FUNCTION_BLOCK changeEventProcess2 (* Basic Function Block Type *)
  (* Standard: 61499-2 *)
  (* Version 0.0, 5/23/2025, azam_w, Schneider Electric, Template *)
  PACKAGE Main;
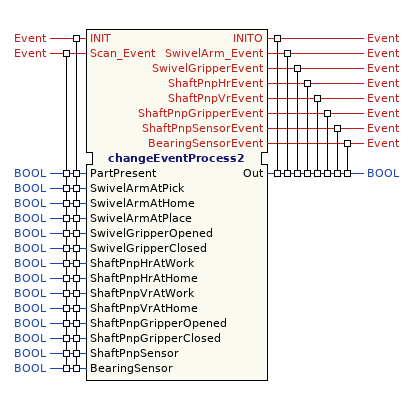
  EVENT_INPUT
    INIT WITH PartPresent, SwivelArmAtPick, SwivelArmAtHome, SwivelArmAtPlace, SwivelGripperOpened, SwivelGripperClosed, ShaftPnpHrAtWork, ShaftPnpHrAtHome, ShaftPnpVrAtWork, ShaftPnpVrAtHome, ShaftPnpGripperOpened, ShaftPnpGripperClosed, ShaftPnpSensor, BearingSensor;
    Scan_Event WITH PartPresent, SwivelArmAtPick, SwivelArmAtHome, SwivelArmAtPlace, SwivelGripperOpened, SwivelGripperClosed, ShaftPnpHrAtWork, ShaftPnpHrAtHome, ShaftPnpVrAtWork, ShaftPnpVrAtHome, ShaftPnpGripperOpened, ShaftPnpGripperClosed, ShaftPnpSensor, BearingSensor;
  END_EVENT
  EVENT_OUTPUT
    INITO WITH Out; (* Initialization Confirm *)
    SwivelArm_Event WITH Out; (* Execution Confirmation *)
    SwivelGripperEvent WITH Out;
    ShaftPnpHrEvent WITH Out;
    ShaftPnpVrEvent WITH Out;
    ShaftPnpGripperEvent WITH Out;
    ShaftPnpSensorEvent WITH Out;
    BearingSensorEvent WITH Out;
  END_EVENT
  VAR_INPUT
    PartPresent : BOOL; (* Output event qualifier *)
    SwivelArmAtPick : BOOL;
    SwivelArmAtHome : BOOL;
    SwivelArmAtPlace : BOOL;
    SwivelGripperOpened : BOOL;
    SwivelGripperClosed : BOOL;
    ShaftPnpHrAtWork : BOOL;
    ShaftPnpHrAtHome : BOOL;
    ShaftPnpVrAtWork : BOOL;
    ShaftPnpVrAtHome : BOOL;
    ShaftPnpGripperOpened : BOOL;
    ShaftPnpGripperClosed : BOOL;
    ShaftPnpSensor : BOOL;
    BearingSensor : BOOL;
  END_VAR
  VAR_OUTPUT
    Out : BOOL;
  END_VAR
  VAR
    PartPresent_PrevVAl : BOOL := FALSE;
    SwivelArmAtPick_PrevVal : BOOL := FALSE;
    SwivelArmAtHome_PrevVal : BOOL := FALSE;
    SwivelArmAtPlace_PrevVal : BOOL := FALSE;
    SwivelGripperClosed_PrevVal : BOOL;
    SwivelGripperOpened_PrevVal : BOOL;
    ShaftPnpHrAtWork_PrevVal : BOOL;
    ShaftPnpHrAtHome_PrevVal : BOOL;
    ShaftPnpVrAtWork_PrevVal : BOOL;
    ShaftPnpVrAtHome_PrevVal : BOOL;
    ShaftPnpGripperClosed_PrevVal : BOOL;
    ShaftPnpGripperOpened_PrevVal : BOOL;
    ShaftPnpSensor_PreVal : BOOL;
    BearingSensor_PreVal : BOOL;
  END_VAR
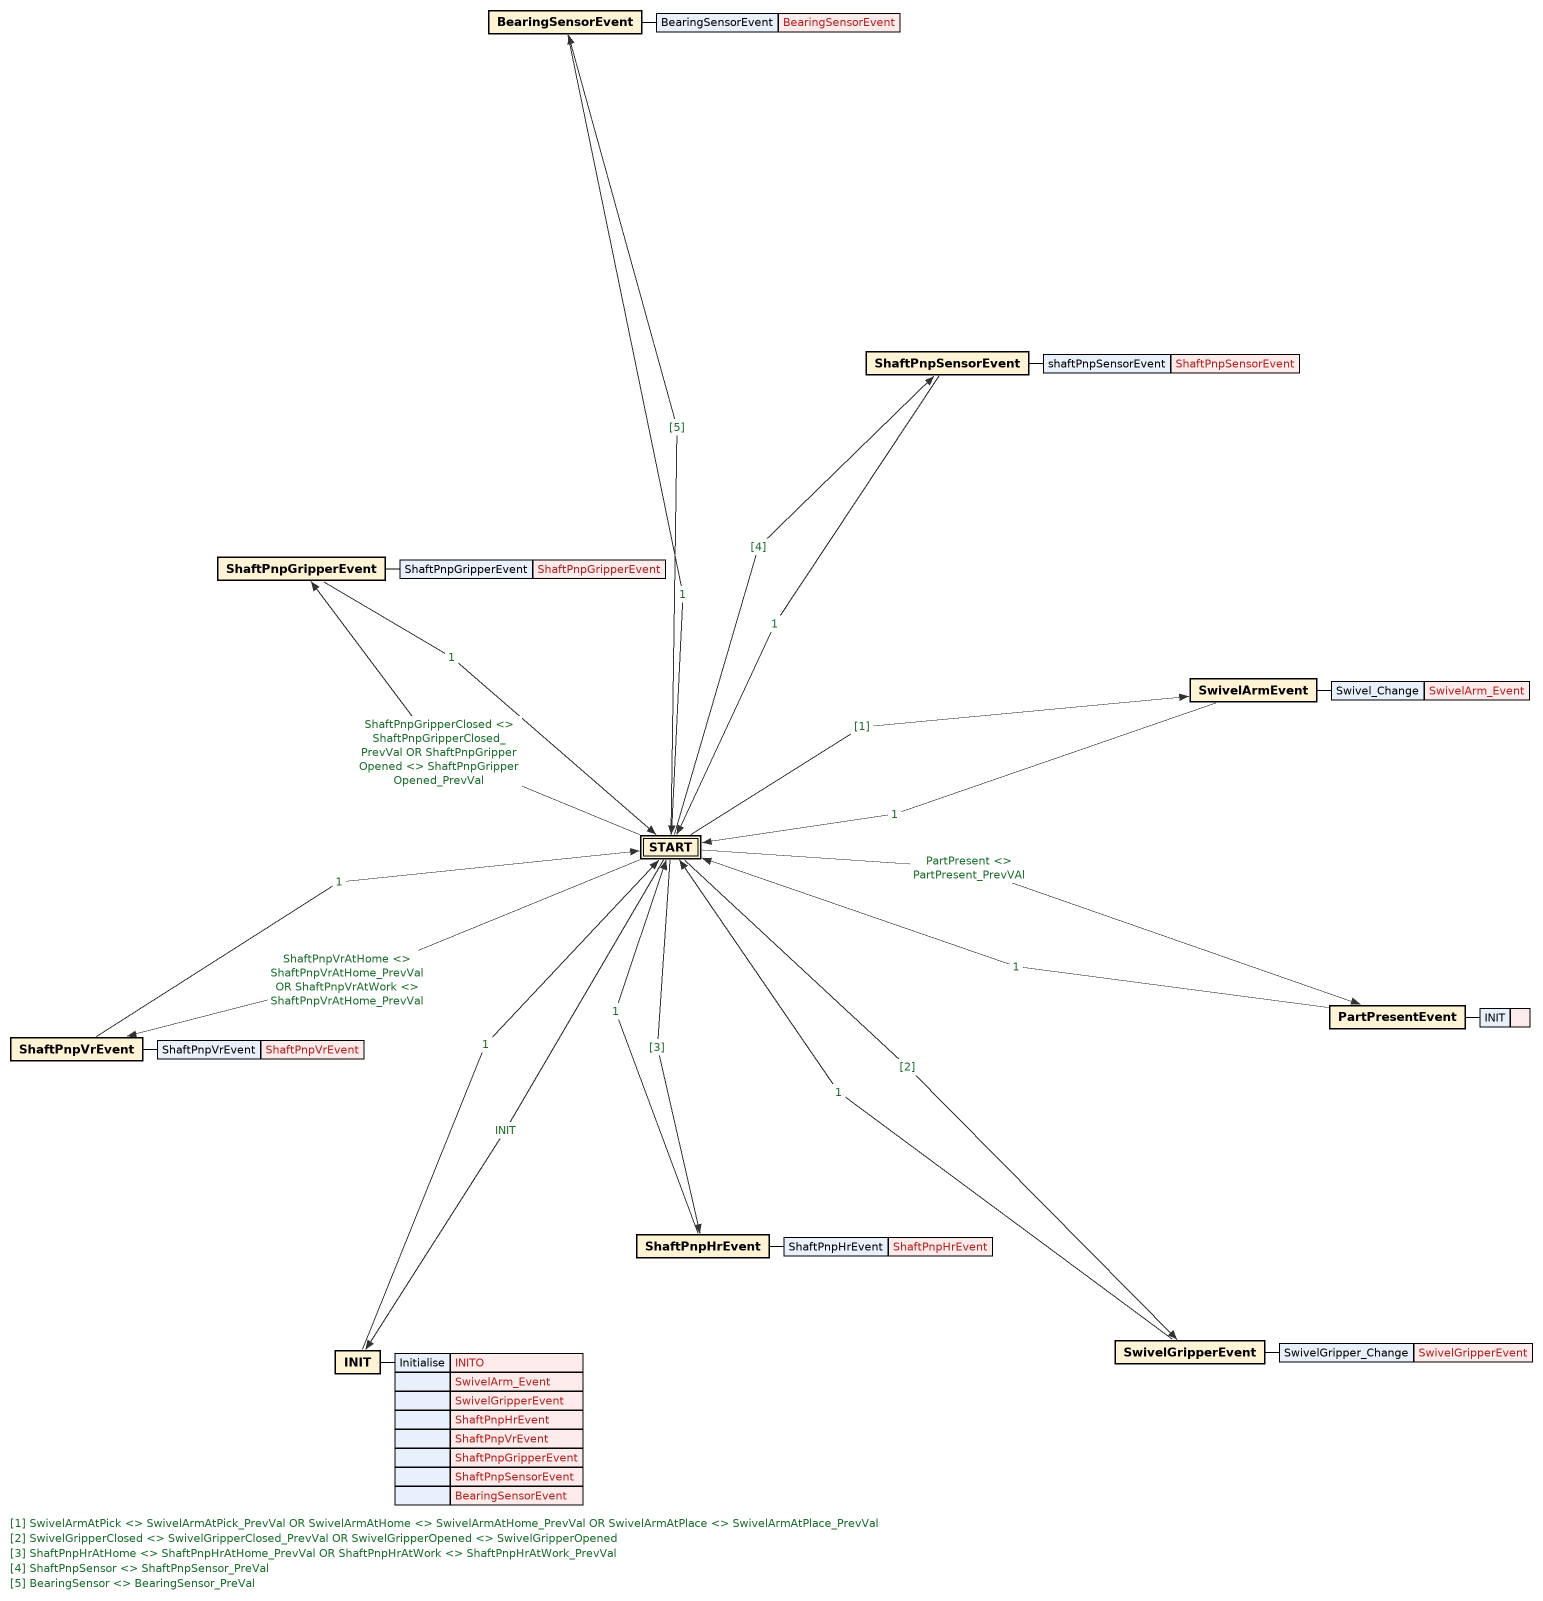
  EC_STATES
    START; (* Initial State *)
    PartPresentEvent : INIT; (* Normal execution *)
    SwivelArmEvent : Swivel_Change -> SwivelArm_Event;
    SwivelGripperEvent : SwivelGripper_Change -> SwivelGripperEvent;
    ShaftPnpHrEvent : ShaftPnpHrEvent -> ShaftPnpHrEvent;
    ShaftPnpVrEvent : ShaftPnpVrEvent -> ShaftPnpVrEvent;
    ShaftPnpGripperEvent : ShaftPnpGripperEvent -> ShaftPnpGripperEvent;
    ShaftPnpSensorEvent : shaftPnpSensorEvent -> ShaftPnpSensorEvent;
    BearingSensorEvent : BearingSensorEvent -> BearingSensorEvent;
    INIT : Initialise -> INITO, -> SwivelArm_Event, -> SwivelGripperEvent, -> ShaftPnpHrEvent, -> ShaftPnpVrEvent, -> ShaftPnpGripperEvent, -> ShaftPnpSensorEvent, -> BearingSensorEvent;
  END_STATES
  EC_TRANSITIONS
    START TO PartPresentEvent := PartPresent <> PartPresent_PrevVAl;
    PartPresentEvent TO START := 1;
    START TO SwivelArmEvent := SwivelArmAtPick <> SwivelArmAtPick_PrevVal OR SwivelArmAtHome <> SwivelArmAtHome_PrevVal OR SwivelArmAtPlace <> SwivelArmAtPlace_PrevVal;
    START TO SwivelGripperEvent := SwivelGripperClosed <> SwivelGripperClosed_PrevVal OR SwivelGripperOpened <> SwivelGripperOpened;
    SwivelGripperEvent TO START := 1;
    START TO ShaftPnpHrEvent := ShaftPnpHrAtHome <> ShaftPnpHrAtHome_PrevVal OR ShaftPnpHrAtWork <> ShaftPnpHrAtWork_PrevVal;
    ShaftPnpHrEvent TO START := 1;
    START TO ShaftPnpVrEvent := ShaftPnpVrAtHome <> ShaftPnpVrAtHome_PrevVal OR ShaftPnpVrAtWork <> ShaftPnpVrAtHome_PrevVal;
    ShaftPnpVrEvent TO START := 1;
    START TO ShaftPnpGripperEvent := ShaftPnpGripperClosed <> ShaftPnpGripperClosed_PrevVal OR ShaftPnpGripperOpened <> ShaftPnpGripperOpened_PrevVal;
    ShaftPnpGripperEvent TO START := 1;
    SwivelArmEvent TO START := 1;
    ShaftPnpSensorEvent TO START := 1;
    START TO ShaftPnpSensorEvent := ShaftPnpSensor <> ShaftPnpSensor_PreVal;
    START TO BearingSensorEvent := BearingSensor <> BearingSensor_PreVal;
    BearingSensorEvent TO START := 1;
    START TO INIT := INIT;
    INIT TO START := 1;
  END_TRANSITIONS
  ALGORITHM INIT IN ST: (* Initialization algorithm *)
;
IF PartPresent <> PartPresent_PrevVAl THEN
	PartPresent_PrevVAl := PartPresent;
	Out := PartPresent;
END_IF;
  END_ALGORITHM
  ALGORITHM Swivel_Change IN ST:
;
IF SwivelArmAtPick <> SwivelArmAtPick_PrevVal THEN
	SwivelArmAtPick_PrevVal := SwivelArmAtPick;
	Out := SwivelArmAtPick;
END_IF;

IF SwivelArmAtHome <> SwivelArmAtHome_PrevVal THEN
	SwivelArmAtHome_PrevVal := SwivelArmAtHome;
	Out := SwivelArmAtHome;
END_IF;

IF SwivelArmAtPlace <> SwivelArmAtPlace_PrevVal THEN
	SwivelArmAtPlace_PrevVal := SwivelArmAtPlace;
	Out := SwivelArmAtPlace;
END_IF;
  END_ALGORITHM
  ALGORITHM SwivelGripper_Change IN ST:
;

IF SwivelGripperOpened <> SwivelGripperOpened_PrevVal THEN
	SwivelGripperOpened_PrevVal := SwivelGripperOpened;
	Out := SwivelGripperOpened;
END_IF;

IF SwivelGripperClosed <> SwivelGripperClosed_PrevVal THEN
	SwivelGripperClosed_PrevVal := SwivelGripperClosed;
	Out := SwivelGripperClosed;
END_IF;
  END_ALGORITHM
  ALGORITHM ShaftPnpHrEvent IN ST:
;
IF ShaftPnpHrAtHome <> ShaftPnpHrAtHome_PrevVal THEN
	ShaftPnpHrAtHome_PrevVal := ShaftPnpHrAtHome;
	Out := ShaftPnpHrAtHome;
END_IF;

IF ShaftPnpHrAtWork <> ShaftPnpHrAtWork_PrevVal THEN
	ShaftPnpHrAtWork_PrevVal := ShaftPnpHrAtWork;
	Out := ShaftPnpHrAtWork;
END_IF;
  END_ALGORITHM
  ALGORITHM ShaftPnpVrEvent IN ST:
;
  END_ALGORITHM
  ALGORITHM ShaftPnpGripperEvent IN ST:
;
  END_ALGORITHM
  ALGORITHM shaftPnpSensorEvent IN ST:
;
IF ShaftPnpSensor <> ShaftPnpSensor_PreVal THEN
	ShaftPnpSensor_PreVal := ShaftPnpSensor;
	Out := ShaftPnpSensor;
END_IF;
  END_ALGORITHM
  ALGORITHM BearingSensorEvent IN ST:
;
IF BearingSensor <> BearingSensor_PreVal THEN
	BearingSensor_PreVal := BearingSensor;
	Out := BearingSensor;
END_IF;
  END_ALGORITHM
  ALGORITHM Initialise IN ST:
Out := TRUE;
  END_ALGORITHM
END_FUNCTION_BLOCK
